FUNCTION_BLOCK Wrapper (* Basic Function Block Type *)
  (* Standard: 61499-2 *)
  (* Version 0.0, 4/9/2019, erik, nxtControl GmbH, Template *)
  PACKAGE Main;
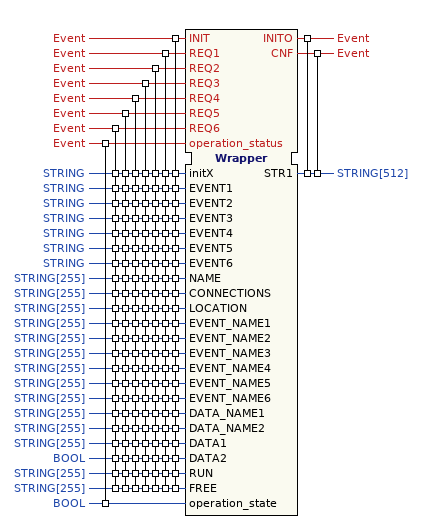
  EVENT_INPUT
    INIT WITH initX, EVENT1, EVENT2, EVENT3, EVENT4, EVENT5, EVENT6, NAME, CONNECTIONS, LOCATION, EVENT_NAME1, EVENT_NAME2, EVENT_NAME3, EVENT_NAME4, EVENT_NAME5, EVENT_NAME6, DATA_NAME1, DATA_NAME2, DATA1, DATA2, RUN, FREE; (* Initialization Request *)
    REQ1 WITH initX, EVENT1, EVENT2, EVENT3, EVENT4, EVENT5, EVENT6, NAME, CONNECTIONS, LOCATION, EVENT_NAME1, EVENT_NAME2, EVENT_NAME3, EVENT_NAME4, EVENT_NAME5, EVENT_NAME6, DATA_NAME1, DATA_NAME2, DATA1, DATA2, RUN, FREE; (* Normal Execution Request *)
    REQ2 WITH initX, EVENT1, EVENT2, EVENT3, EVENT4, EVENT5, EVENT6, NAME, CONNECTIONS, LOCATION, EVENT_NAME1, EVENT_NAME2, EVENT_NAME3, EVENT_NAME4, EVENT_NAME5, EVENT_NAME6, DATA_NAME1, DATA_NAME2, DATA1, DATA2, RUN, FREE;
    REQ3 WITH initX, EVENT1, EVENT2, EVENT3, EVENT4, EVENT5, EVENT6, NAME, CONNECTIONS, LOCATION, EVENT_NAME1, EVENT_NAME2, EVENT_NAME3, EVENT_NAME4, EVENT_NAME5, EVENT_NAME6, DATA_NAME1, DATA_NAME2, DATA1, DATA2, RUN, FREE;
    REQ4 WITH initX, EVENT1, EVENT2, EVENT3, EVENT4, EVENT5, EVENT6, NAME, CONNECTIONS, LOCATION, EVENT_NAME1, EVENT_NAME2, EVENT_NAME3, EVENT_NAME4, EVENT_NAME5, EVENT_NAME6, DATA_NAME1, DATA_NAME2, DATA1, DATA2, RUN, FREE;
    REQ5 WITH initX, EVENT1, EVENT2, EVENT3, EVENT4, EVENT5, EVENT6, NAME, CONNECTIONS, LOCATION, EVENT_NAME1, EVENT_NAME2, EVENT_NAME3, EVENT_NAME4, EVENT_NAME5, EVENT_NAME6, DATA_NAME1, DATA_NAME2, DATA1, DATA2, RUN, FREE;
    REQ6 WITH initX, EVENT1, EVENT2, EVENT3, EVENT4, EVENT5, EVENT6, NAME, CONNECTIONS, LOCATION, EVENT_NAME1, EVENT_NAME2, EVENT_NAME3, EVENT_NAME4, EVENT_NAME5, EVENT_NAME6, DATA_NAME1, DATA_NAME2, DATA1, DATA2, RUN, FREE;
    operation_status WITH operation_state;
  END_EVENT
  EVENT_OUTPUT
    INITO WITH STR1; (* Initialization Confirm *)
    CNF WITH STR1; (* Execution Confirmation *)
  END_EVENT
  VAR_INPUT
    initX : STRING;
    EVENT1 : STRING;
    EVENT2 : STRING;
    EVENT3 : STRING;
    EVENT4 : STRING;
    EVENT5 : STRING;
    EVENT6 : STRING;
    NAME : STRING[255];
    CONNECTIONS : STRING[255];
    LOCATION : STRING[255];
    EVENT_NAME1 : STRING[255];
    EVENT_NAME2 : STRING[255];
    EVENT_NAME3 : STRING[255];
    EVENT_NAME4 : STRING[255];
    EVENT_NAME5 : STRING[255];
    EVENT_NAME6 : STRING[255];
    DATA_NAME1 : STRING[255];
    DATA_NAME2 : STRING[255];
    DATA1 : STRING[255];
    DATA2 : BOOL;
    RUN : STRING[255];
    FREE : STRING[255];
    operation_state : BOOL;
  END_VAR
  VAR_OUTPUT
    STR1 : STRING[512]; (* Output event qualifier *)
  END_VAR
  VAR
    Global_var1 : INT;
    text1 : STRING[255];
  END_VAR
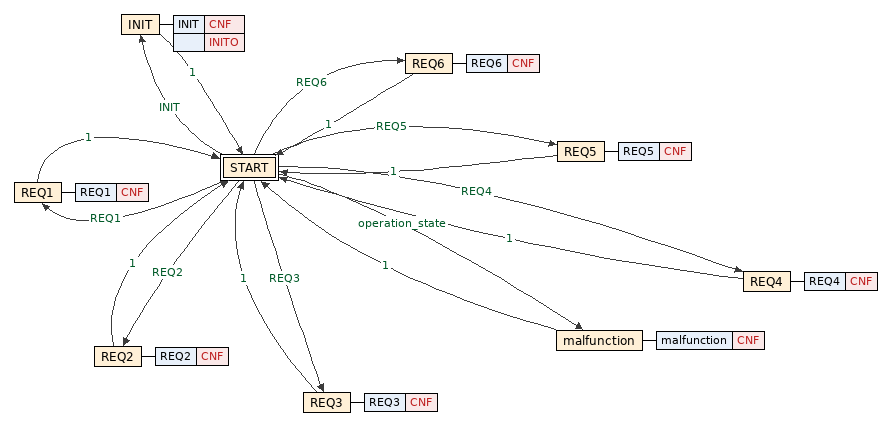
  EC_STATES
    START; (* Initial State *)
    INIT : INIT -> CNF, -> INITO; (* Initialization *)
    REQ1 : REQ1 -> CNF; (* Normal execution *)
    REQ2 : REQ2 -> CNF;
    REQ3 : REQ3 -> CNF;
    REQ4 : REQ4 -> CNF;
    REQ5 : REQ5 -> CNF;
    REQ6 : REQ6 -> CNF;
    malfunction : malfunction -> CNF;
  END_STATES
  EC_TRANSITIONS
    START TO INIT := INIT;
    INIT TO START := 1;
    START TO REQ1 := REQ1;
    START TO REQ2 := REQ2;
    START TO REQ3 := REQ3;
    REQ1 TO START := 1;
    REQ3 TO START := 1;
    REQ2 TO START := 1;
    REQ4 TO START := 1;
    START TO REQ4 := REQ4;
    START TO REQ5 := REQ5;
    REQ5 TO START := 1;
    START TO REQ6 := REQ6;
    REQ6 TO START := 1;
    START TO malfunction := operation_state;
    malfunction TO START := 1;
  END_TRANSITIONS
  ALGORITHM INIT IN ST: (* Initialization algorithm *)
VAR
	text : STRING[255];
  events : STRING[255];
  data : STRING[255];
  len1 : DINT;
END_VAR

Global_var1 := 0;
events := '';
text := '';

(*target is: initi;name;event:event1;data1:data2;location;connections;%event:event1;data1:data2;*)
(*target is: inito;name;event:event1;data1:data2;*)

(*initX is the type of init and IN_STR1 is the name*)
STR1 := initX;
STR1 := CONCAT(STR1,';');
STR1 := CONCAT(STR1,NAME);
STR1 := CONCAT(STR1,';');

IF initX = 'initi' THEN
  (*EVENT_NAME1 - EVENT_NAME5 are the events/methods for the hardware model*)
  IF EVENT_NAME1 <> '' THEN
  	events := CONCAT(events,EVENT_NAME1);
  	events := CONCAT(events,':');
  END_IF;
  IF EVENT_NAME2 <> '' THEN
  	events := CONCAT(events,EVENT_NAME2);
  	events := CONCAT(events,':');
  END_IF;
  IF EVENT_NAME3 <> '' THEN
  	events := CONCAT(events,EVENT_NAME3);
  	events := CONCAT(events,':');
  END_IF;
  IF EVENT_NAME4 <> '' THEN
  	events := CONCAT(events,EVENT_NAME4);
  	events := CONCAT(events,':');
  END_IF;
  IF EVENT_NAME5 <> '' THEN
  	events := CONCAT(events,EVENT_NAME5);
  	events := CONCAT(events,':');
  END_IF;
  IF EVENT_NAME6 <> '' THEN
	  events := CONCAT(events,EVENT_NAME6);
	  events := CONCAT(events,':');
  END_IF;
  IF events <> '' THEN
  	len1 := LEN(events);
  	events := LEFT(events, len1 -1);
  END_IF;
  events := CONCAT(events, ';');

  (*joining the events to the STR1*)
  STR1 := CONCAT(STR1, events);

  (*location*)
	IF LOCATION <> '' THEN
		STR1 := CONCAT(STR1, LOCATION);
	ELSE
		STR1 := CONCAT(STR1,'None');
	END_IF;
	STR1 := CONCAT(STR1, ';');

	(*connections*)
	IF CONNECTIONS <> '' THEN
		STR1 := CONCAT(STR1, CONNECTIONS);
	ELSE
		STR1 := CONCAT(STR1,'None');
	END_IF;
	STR1 := CONCAT(STR1, ';');

	(*hardware and fb model split here*)
	STR1 := CONCAT(STR1, '%');
END_IF;

(*events for fb model*)
events := '';
IF EVENT1 <> '' THEN
	events := CONCAT(events,EVENT1);
	events := CONCAT(events,':');
END_IF;
IF EVENT2 <> '' THEN
	events := CONCAT(events,EVENT2);
	events := CONCAT(events,':');
END_IF;
IF EVENT3 <> '' THEN
	events := CONCAT(events,EVENT3);
	events := CONCAT(events,':');
END_IF;
IF EVENT4 <> '' THEN
	events := CONCAT(events,EVENT4);
	events := CONCAT(events,':');
END_IF;
IF EVENT5 <> '' THEN
	events := CONCAT(events,EVENT5);
	events := CONCAT(events,':');
END_IF;
IF EVENT6 <> '' THEN
	events := CONCAT(events,EVENT6);
	events := CONCAT(events,':');
END_IF;
IF events <> '' THEN
	len1 := LEN(events);
	events := LEFT(events, len1 -1);
END_IF;
events := CONCAT(events, ';');

(*joining events to str1*)
STR1 := CONCAT(STR1,events);

(*data*)
data := '';
IF DATA_NAME1 <> '' THEN
	data := CONCAT(data,DATA1);
	data := CONCAT(data,':');
END_IF;
(*data2 is bool*)
(*this is not finished yet, might cause errors at opc side, since opc is only waiting name of the data*)
(*IF DATA_NAME2 <> '' THEN
  data := CONCAT(data,DATA_NAME2);
  data := CONCAT(data,'=');
	IF DATA2 <> FALSE THEN
		data := CONCAT(data,'TRUE');
	ELSE
		data := CONCAT(data,'FALSE');
	END_IF;
	data := CONCAT(data,':');
END_IF;*)
IF data <> '' THEN
	len1 := LEN(data);
	data := LEFT(data, len1 -1);
END_IF;

data := CONCAT(data, ';');


(*joining data to STR1*)
STR1 := CONCAT(STR1,data);
  END_ALGORITHM
  ALGORITHM REQ1 IN ST: (* Normally executed algorithm *)
;
text1 := '';
IF FIND(FREE,'REQ1') <> 0 THEN
  text1 := 'Free';
END_IF;

IF FIND(RUN,'REQ1') <> 0 THEN
  text1 := 'Running';
END_IF;

Global_var1 := 1;



STR1 := CONCAT('update;',NAME);
STR1 := CONCAT(STR1,';');

STR1 := CONCAT(STR1,EVENT1);
STR1 := CONCAT(STR1,';');
IF text1 <> '' THEN
	STR1 := CONCAT(STR1,text1);
ELSE
	STR1 := CONCAT(STR1,'None');
END_IF;
STR1 := CONCAT(STR1,';');
  END_ALGORITHM
  ALGORITHM REQ2 IN ST:
;
text1 := '';
IF FIND(FREE,'REQ2')<> 0  THEN
  text1 := 'Free';
END_IF;

IF FIND(RUN,'REQ2') <> 0 THEN
  text1 := 'Running';
END_IF;
Global_var1 := 2;


STR1 := CONCAT('update;',NAME);
STR1 := CONCAT(STR1,';');

STR1 := CONCAT(STR1,EVENT2);
STR1 := CONCAT(STR1,';');

IF text1 <> '' THEN
	STR1 := CONCAT(STR1,text1);
ELSE
	STR1 := CONCAT(STR1,'None');
END_IF;
STR1 := CONCAT(STR1,';');
  END_ALGORITHM
  ALGORITHM REQ3 IN ST:
;
text1 := '';
IF FIND(FREE,'REQ3') <> 0 THEN
  text1 := 'Free';
END_IF;

IF FIND(RUN,'REQ3') <> 0 THEN
  text1 := 'Running';
END_IF;
Global_var1 := 3;


STR1 := CONCAT('update;',NAME);
STR1 := CONCAT(STR1,';');

STR1 := CONCAT(STR1,EVENT3);
STR1 := CONCAT(STR1,';');

IF text1 <> '' THEN
	STR1 := CONCAT(STR1,text1);
ELSE
	STR1 := CONCAT(STR1,'None');
END_IF;
STR1 := CONCAT(STR1,';');
  END_ALGORITHM
  ALGORITHM REQ4 IN ST:
;
text1 := '';
IF FIND(FREE,'REQ4') <> 0 THEN
  text1 := 'Free';
END_IF;

IF FIND(RUN,'REQ4') <> 0 THEN
  text1 := 'Running';
END_IF;
Global_var1 := 4;


STR1 := CONCAT('update;',NAME);
STR1 := CONCAT(STR1,';');

STR1 := CONCAT(STR1,EVENT4);
STR1 := CONCAT(STR1,';');

IF text1 <> '' THEN
	STR1 := CONCAT(STR1,text1);
ELSE
	STR1 := CONCAT(STR1,'None');
END_IF;
STR1 := CONCAT(STR1,';');
  END_ALGORITHM
  ALGORITHM REQ5 IN ST:
;
text1 := '';
IF FIND(FREE,'REQ5') <> 0 THEN
  text1 := 'Free';
END_IF;

IF FIND(RUN,'REQ5') <> 0 THEN
  text1 := 'Running';
END_IF;
Global_var1 := 5;


STR1 := CONCAT('update;',NAME);
STR1 := CONCAT(STR1,';');

STR1 := CONCAT(STR1,EVENT5);
STR1 := CONCAT(STR1,';');

IF text1 <> '' THEN
	STR1 := CONCAT(STR1,text1);
ELSE
	STR1 := CONCAT(STR1,'None');
END_IF;
STR1 := CONCAT(STR1,';');
  END_ALGORITHM
  ALGORITHM REQ6 IN ST:
;
text1 := '';
IF FIND(FREE,'REQ6') <> 0 THEN
  text1 := 'Free';
END_IF;

IF FIND(RUN,'REQ6') <> 0 THEN
  text1 := 'Running';
END_IF;
Global_var1 := 5;


STR1 := CONCAT('update;',NAME);
STR1 := CONCAT(STR1,';');

STR1 := CONCAT(STR1,EVENT6);
STR1 := CONCAT(STR1,';');

IF text1 <> '' THEN
	STR1 := CONCAT(STR1,text1);
ELSE
	STR1 := CONCAT(STR1,'None');
END_IF;
STR1 := CONCAT(STR1,';');
  END_ALGORITHM
  ALGORITHM malfunction IN ST:
;


STR1 := CONCAT('update;',NAME);
STR1 := CONCAT(STR1,';');

//STR1 := CONCAT(STR1,EVENT?);
STR1 := CONCAT(STR1,';');

IF operation_state = TRUE THEN
	STR1 := CONCAT(STR1,'Free');
ELSE
	STR1 := CONCAT(STR1,'Malfunctioning');
END_IF;
STR1 := CONCAT(STR1,';');
  END_ALGORITHM
END_FUNCTION_BLOCK
